PROGRAM MAIN

VAR
	
	
	bGreenBtn    : POINTER TO BOOL:= ADR(GVL_IO.aInputs[1]);
	bRedBtn		: POINTER TO BOOL:= ADR(GVL_IO.aInputs[2]);
	bLight : POINTER TO BOOL := ADR(GVL_IO.aOutputs[1]);

	fbStartInput : fbDigitalInput(ioBitRef := ADR(GVL_IO.aInputs[1]), switchType := E_SwitchType.NO);
	fbStopInput : fbDigitalInput(ioBitRef := ADR(GVL_IO.aInputs[2]), switchType := E_SwitchType.NC);
	fbLightOutput : fbDigitalOutput(ioBitRef := ADR(GVL_IO.aOutputs[1]), switchType := E_SwitchType.NO);
	light2 : fbDigitalOutput(ioBitRef := ADR(GVL_IO.aOutputs[2]), switchType := E_SwitchType.NO);
	CurrentState: UINT  := TO_UINT(E_LightStates.FAST_BLINK);
	
	fbCounter : CTU;

	timedLight : BOOL;
	timer :TON;

	aLightCurtain : ARRAY[1..10] OF BOOL; 
	
	myPisa : FB_PISA_Comms(sProductName := 'PISA-M-4CL2');
	
	cbStates : ARRAY[1..4] OF CircuitBreakerStatus;
	i: INT;
END_VAR




GVL_IO.aOutputs[8] := GVL_IO.aInputs[8]; // Output 8 mirrors input 8


IF fbStartInput.Get() THEN
		fbLightOutput.Set(TRUE);
ELSE 
		fbLightOutput.Set(FALSE);
END_IF

//bGreenBtn := aInputs[1];


(*
IF bGreenBtn^ THEN
		bLight^:=TRUE;
ELSE 
		bLight^:=FALSE;
END_IF
*)
myPisa();

FOR i := 1 TO 4 DO
    cbStates[i] := myPisa.GetStatus(i);
END_FOR;

fbCounter(CU:=fbStartInput.Get(),CU:=fbStartInput.Get(), RESET :=fbStopInput.Get() ,PV := UINT_TO_WORD(E_LightStates.COUNT));
CurrentState:=fbCounter.CV;


	aLightCurtain[1]:= (GVL_IO.flexChain.pdo[GVL_IO.lightBarPDOstartIndex] AND 2#0000_0000_0000_0001) <> 0;
	aLightCurtain[2]:= (GVL_IO.flexChain.pdo[GVL_IO.lightBarPDOstartIndex] AND 2#0000_0000_0000_0010) <> 0;
	aLightCurtain[3]:= (GVL_IO.flexChain.pdo[GVL_IO.lightBarPDOstartIndex] AND 2#0000_0000_0000_0100) <> 0;
	aLightCurtain[4]:= (GVL_IO.flexChain.pdo[GVL_IO.lightBarPDOstartIndex] AND 2#0000_0000_0000_1000) <> 0;
	aLightCurtain[5]:= (GVL_IO.flexChain.pdo[GVL_IO.lightBarPDOstartIndex] AND 2#0000_0000_0001_0000) <> 0;
	aLightCurtain[6]:= (GVL_IO.flexChain.pdo[GVL_IO.lightBarPDOstartIndex] AND 2#0000_0000_0010_0000) <> 0;
	aLightCurtain[7]:= (GVL_IO.flexChain.pdo[GVL_IO.lightBarPDOstartIndex] AND 2#0000_0000_0100_0000) <> 0;
	aLightCurtain[8]:= (GVL_IO.flexChain.pdo[GVL_IO.lightBarPDOstartIndex] AND 2#0000_0000_1000_0000) <> 0;
	aLightCurtain[9]:= (GVL_IO.flexChain.pdo[GVL_IO.lightBarPDOsecondIndex] AND 2#0000_0000_0000_0001) <> 0;
	aLightCurtain[10]:= (GVL_IO.flexChain.pdo[GVL_IO.lightBarPDOsecondIndex] AND 2#0000_0000_0000_0010) <> 0;
								


CASE CurrentState OF
    E_LightStates.OFF:
		fbLightOutput.Set(FALSE);
    E_LightStates.ON:
		fbLightOutput.Set(TRUE);
    E_LightStates.SLOW_BLINK:
		timer(IN := NOT timer.Q, PT := T#1S500MS);
		IF timer.Q THEN 
			timedLight := NOT timedLight; 
		END_IF
		fbLightOutput.Set(timedLight);
    E_LightStates.FAST_BLINK:
		timer(IN := NOT timer.Q, PT := T#0S500MS);
		IF timer.Q THEN 
			timedLight := NOT timedLight; 
		END_IF
		fbLightOutput.Set(timedLight);
ELSE
		fbLightOutput.Set(FALSE);
		fbCounter(RESET:=TRUE);
		
END_CASE

IF GVL_IO.Encoder_Counts > 500 THEN
	light2.Set(TRUE);
ELSE
	light2.Set(FALSE);		

END_IF

END_PROGRAM

(* stored: Version 1.1.0.1, ProductVersion 3.1.4024.15
   POU MAIN: Id {2619c018-a97e-4e98-bfde-76b022b13f51}, SpecialFunc None *)
